INTERFACE INTERNAL I_StateAdapter

PROPERTY INTERNAL _AsIStateInternal : I_StateInternal
GET
END_GET
END_PROPERTY

END_INTERFACE

(* stored: Version 1.1.0.1
   Itf I_StateAdapter: Id {fd9fce22-961d-496b-90f4-a68f24247074}
   Property _AsIStateInternal: Id {6ba7e1ce-ccfb-4966-b3ab-4e2927f81551}
   Get Get: Id {b2766e60-6c6f-4835-a2fa-4210a114d499} *)
